FUNCTION_BLOCK Model (* Composite Function Block Type *)
  (* Standard: 61499-2 *)
  (* Version 0.0, 2/7/2012, XPMUser, nxtControl GmbH, template *)
  PACKAGE Main;
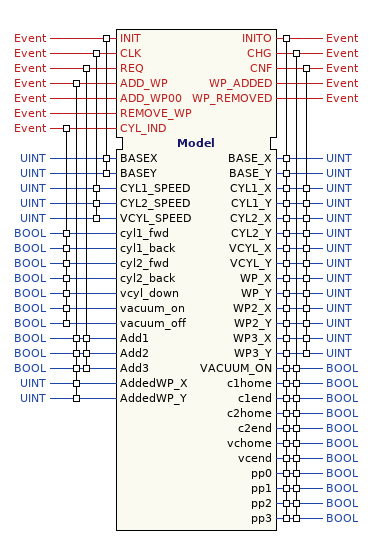
  EVENT_INPUT
    INIT WITH BASEX, BASEY; (* Initialization Request *)
    CLK WITH CYL1_SPEED, CYL2_SPEED, VCYL_SPEED; (* Clock *)
    REQ WITH Add1, Add2, Add3;
    ADD_WP WITH Add1, Add2, Add3, AddedWP_X, AddedWP_Y;
    ADD_WP00;
    REMOVE_WP;
    CYL_IND WITH cyl1_fwd, cyl1_back, cyl2_fwd, cyl2_back, vcyl_down, vacuum_on, vacuum_off;
  END_EVENT
  EVENT_OUTPUT
    INITO WITH BASE_X, BASE_Y, CYL1_X, CYL1_Y, CYL2_X, CYL2_Y, VCYL_X, VCYL_Y, WP_X, WP_Y, WP2_X, WP2_Y, WP3_X, WP3_Y, VACUUM_ON, c1home, c1end, c2home, c2end, vchome, vcend, pp0, pp1, pp2, pp3; (* Initialization Confirm *)
    CHG WITH c1home, c1end, c2home, c2end, vchome, vcend, pp0, pp1, pp2, pp3, VACUUM_ON; (* View State Changed *)
    CNF WITH VCYL_Y, WP_X, WP_Y, WP2_X, WP2_Y, WP3_X, WP3_Y, CYL2_X, VCYL_X, CYL2_Y, CYL1_Y, CYL1_X;
    WP_ADDED;
    WP_REMOVED;
  END_EVENT
  VAR_INPUT
    BASEX : UINT;
    BASEY : UINT;
    CYL1_SPEED : UINT;
    CYL2_SPEED : UINT;
    VCYL_SPEED : UINT;
    cyl1_fwd : BOOL;
    cyl1_back : BOOL; (* Response Data from Socket *)
    cyl2_fwd : BOOL;
    cyl2_back : BOOL;
    vcyl_down : BOOL;
    vacuum_on : BOOL;
    vacuum_off : BOOL;
    Add1 : BOOL;
    Add2 : BOOL;
    Add3 : BOOL;
    AddedWP_X : UINT;
    AddedWP_Y : UINT;
  END_VAR
  VAR_OUTPUT
    BASE_X : UINT; (* Response Data from Socket *)
    BASE_Y : UINT; (* Response Data from Socket *)
    CYL1_X : UINT; (* Response Data from Socket *)
    CYL1_Y : UINT; (* Response Data from Socket *)
    CYL2_X : UINT; (* Response Data from Socket *)
    CYL2_Y : UINT; (* Response Data from Socket *)
    VCYL_X : UINT; (* Response Data from Socket *)
    VCYL_Y : UINT; (* Response Data from Socket *)
    WP_X : UINT; (* Response Data from Socket *)
    WP_Y : UINT; (* Response Data from Socket *)
    WP2_X : UINT; (* Response Data from Socket *)
    WP2_Y : UINT; (* Response Data from Socket *)
    WP3_X : UINT; (* Response Data from Socket *)
    WP3_Y : UINT; (* Response Data from Socket *)
    VACUUM_ON : BOOL; (* Response Data from Socket *)
    c1home : BOOL;
    c1end : BOOL;
    c2home : BOOL;
    c2end : BOOL;
    vchome : BOOL;
    vcend : BOOL;
    pp0 : BOOL;
    pp1 : BOOL;
    pp2 : BOOL;
    pp3 : BOOL;
  END_VAR
  FBS
    WPSensors : WP_Sensor;
    ViewControl : PnpXYCalculator;
    FB2 : OutputSender;
    FB1 : InputSender;
    Cylinder : PnpCylinders(InitialPosition := 0.0, HomeSensorRange := [0,0], MidSensorRange := [50,50], EndSensorRange := [100,100], Loaded := 0, LoadType := 0, LCMovingtDistance := 75, RCMovingtDistance := 150, VCMovingtDistance := 75);
    SuctionUnit : PnPVacuum;
  END_FBS
  EVENT_CONNECTIONS
    ADD_WP TO ViewControl.ADD_WP;
    ADD_WP00 TO ViewControl.ADD_WP00;
    REMOVE_WP TO ViewControl.REMOVE_WP;
    ViewControl.WP_ADDED TO WP_ADDED;
    ViewControl.WP_REMOVED TO WP_REMOVED;
    Cylinder.INITO TO SuctionUnit.INIT;
    SuctionUnit.INITO TO ViewControl.INIT;
    SuctionUnit.CHG TO ViewControl.CLK;
    ViewControl.INITO TO WPSensors.INIT;
    WPSensors.CNF TO CHG;
    WPSensors.INITO TO INITO;
    ViewControl.CNF TO WPSensors.REQ;
    Cylinder.CNF TO ViewControl.CLK;
    Cylinder.CHG TO CHG;
    SuctionUnit.CHG TO CHG;
    ViewControl.CNF TO CNF;
    CYL_IND TO ViewControl.REQ;
    FB1.RESET TO Cylinder.RESET;
    Cylinder.INITO TO FB2.INIT;
    INIT TO FB1.INIT;
    FB1.INITO TO Cylinder.INIT;
    FB2.CNF TO FB1.REQ;
    FB1.CNF TO Cylinder.CLK;
    REQ TO FB1.REQ;
    Cylinder.CHG_RESET TO SuctionUnit.RESET;
    SuctionUnit.CHG_RESET TO FB2.REQ;
    Cylinder.CHG TO SuctionUnit.CLK;
    SuctionUnit.CHG TO FB2.REQ;
  END_CONNECTIONS
  DATA_CONNECTIONS
    ViewControl.BASE_X TO BASE_X;
    ViewControl.BASE_Y TO BASE_Y;
    ViewControl.WP_X TO WP_X;
    ViewControl.WP_Y TO WP_Y;
    ViewControl.WP2_X TO WP2_X;
    ViewControl.WP2_Y TO WP2_Y;
    ViewControl.WP3_X TO WP3_X;
    ViewControl.WP3_Y TO WP3_Y;
    BASEX TO ViewControl.BASEX;
    BASEY TO ViewControl.BASEY;
    Add1 TO ViewControl.Add1;
    Add2 TO ViewControl.Add2;
    Add3 TO ViewControl.Add3;
    AddedWP_X TO ViewControl.AddedWP_X;
    AddedWP_Y TO ViewControl.AddedWP_Y;
    Cylinder.LCAbsolutePos TO ViewControl.LCPos;
    CYL1_SPEED TO Cylinder.LCForwardSpeed;
    CYL1_SPEED TO Cylinder.LCBackwardSpeed;
    CYL2_SPEED TO Cylinder.RCForwardSpeed;
    CYL2_SPEED TO Cylinder.RCBackwardSpeed;
    VCYL_SPEED TO Cylinder.VCSpeed;
    Cylinder.RCAbsolutePos TO ViewControl.RCPos;
    Cylinder.VCAbsolutePos TO ViewControl.VCPos;
    SuctionUnit.VacState TO ViewControl.vacuumon;
    ViewControl.WP_X TO WPSensors.WP1_X;
    ViewControl.WP_Y TO WPSensors.WP1_Y;
    ViewControl.WP2_X TO WPSensors.WP2_X;
    ViewControl.WP2_Y TO WPSensors.WP2_Y;
    ViewControl.WP3_X TO WPSensors.WP3_X;
    ViewControl.WP3_Y TO WPSensors.WP3_Y;
    WPSensors.wp11 TO pp0;
    WPSensors.wp14 TO pp3;
    WPSensors.wp13 TO pp2;
    WPSensors.wp12 TO pp1;
    cyl1_fwd TO FB1.cyl1_fwd;
    FB1.c1extend TO Cylinder.LCExtend;
    cyl1_back TO FB1.cyl1_back;
    FB1.c1retract TO Cylinder.LCRetract;
    cyl2_fwd TO FB1.cyl2_fwd;
    FB1.c2extend TO Cylinder.RCExtend;
    cyl2_back TO FB1.cyl2_back;
    FB1.c2retract TO Cylinder.RCRetract;
    vacuum_on TO FB1.vacuum_on;
    FB1.vacuumOn TO SuctionUnit.VacuumOn;
    FB1.vacuumOn TO ViewControl.vacuum_on;
    vacuum_off TO FB1.vacuum_off;
    FB1.vacuumOff TO SuctionUnit.VacuumOff;
    FB1.vacuumOff TO ViewControl.vacuum_off;
    vcyl_down TO FB1.vcyl_down;
    FB1.vcxtend TO Cylinder.VCExtend;
    SuctionUnit.VacState TO FB2.VACUUM_ON;
    FB2.vacuum_on TO VACUUM_ON;
    Cylinder.LCAtHome TO FB2.c1home;
    FB2.c1_home TO c1home;
    Cylinder.LCAtEnd TO FB2.c1end;
    FB2.c1_end TO c1end;
    Cylinder.RCAtHome TO FB2.c2home;
    FB2.c2_home TO c2home;
    Cylinder.RCAtEnd TO FB2.c2end;
    FB2.c2_end TO c2end;
    Cylinder.VCAtHome TO FB2.vchome;
    FB2.vc_home TO vchome;
    Cylinder.VCAtEnd TO FB2.vcend;
    FB2.vc_end TO vcend;
    FB1.resetVACUUM_ON TO SuctionUnit.resetVacuumOn;
    FB1.resetC1home TO Cylinder.resetLCAtHome;
    FB1.resetC1end TO Cylinder.resetLCAtEnd;
    FB1.resetC2home TO Cylinder.resetRCAtHome;
    FB1.resetC2end TO Cylinder.resetRCAtEnd;
    FB1.resetVChome TO Cylinder.resetVCAtHome;
    FB1.resetVCend TO Cylinder.resetVCAtEnd;
    ViewControl.CYL1_X TO CYL1_X;
    ViewControl.CYL1_Y TO CYL1_Y;
    ViewControl.CYL2_X TO CYL2_X;
    ViewControl.CYL2_Y TO CYL2_Y;
    ViewControl.VCYL_X TO VCYL_X;
    ViewControl.VCYL_Y TO VCYL_Y;
    FB1.resetC1AbsPos TO Cylinder.resetC1AbsPos;
    FB1.resetC2AbsPos TO Cylinder.resetC2AbsPos;
    FB1.resetVCAbsPos TO Cylinder.resetVCAbsPos;
    Cylinder.RCAbsolutePos TO FB2.c2AbsPos;
    Cylinder.LCAbsolutePos TO FB2.c1AbsPos;
    Cylinder.VCAbsolutePos TO FB2.vcAncPos;
  END_CONNECTIONS
END_FUNCTION_BLOCK
